# B&R Automation Studio project turbo-parakeet-aka-lab_3
Automation Studio 

## Logical view

### Global.var
```iecst
VAR
	AxisX : ACP10AXIS_typ := (0);
	AxisX_EncIf : SdcEncIf16_typ := (0);
	AxisX_DrvIf : SdcDrvIf16_typ := (0);
	AxisX_DiDoIf : SdcDiDoIf_typ := (0);
	AxisX_HW : SdcHwCfg_typ := (0);
	AxisY : ACP10AXIS_typ := (0);
	AxisY_EncIf : SdcEncIf16_typ := (0);
	AxisY_DrvIf : SdcDrvIf16_typ := (0);
	AxisY_DiDoIf : SdcDiDoIf_typ := (0);
	AxisY_HW : SdcHwCfg_typ := (0);
	AxisZ : ACP10AXIS_typ := (0);
	AxisZ_EncIf : SdcEncIf16_typ := (0);
	AxisZ_DrvIf : SdcDrvIf16_typ := (0);
	AxisZ_DiDoIf : SdcDiDoIf_typ := (0);
	AxisZ_HW : SdcHwCfg_typ := (0);
	gAxis01 : ACP10AXIS_typ := (0);
	gAxis02 : ACP10AXIS_typ := (0);
	gAxisTest : ACP10AXIS_typ := (0);
	gAxisTest_HW : SdcHwCfg_typ := (0);
	gAxisTest_DrvIf : SdcDrvIf16_typ := (0);
	gAxisTest_DiDoIf : SdcDiDoIf_typ := (0);
	gAxisTest_ModuleOk : BOOL := 0;
	gAxis03 : ACP10AXIS_typ := (0);
	gAxis03_HW : SdcHwCfg_typ := (0);
	gAxis03_DrvIf : SdcDrvIf16_typ := (0);
	gAxis03_DiDoIf : SdcDiDoIf_typ := (0);
	gAxis03_ModuleOk : BOOL := 0;
	CNCsys : ARNC0CNC_typ;
	position : INT := 0;
	Myspeed : INT := 0;
END_VAR
```

### Program Logical/SDCAxisCtr

#### Main.c
```c
#include <bur/plctypes.h>

#ifdef _DEFAULT_INCLUDES
	#include <AsDefault.h>
#endif

void increase_counters(void);

void _INIT ProgramInit(void)
{
	//Устанваливаем типы SDC модулей
	AxisX_HW.EncIf1_Typ = ncSDC_ENC16;
	AxisX_HW.DiDoIf_Typ = ncSDC_DIDO;
	AxisX_HW.DrvIf_Typ = ncSDC_DRVSERVO16;

	//Устанавливаем имена переменных
	strcpy(AxisX_HW.EncIf1_Name, "AxisX_EncIf");
	strcpy(AxisX_HW.DrvIf_Name, "AxisX_DrvIf");
	strcpy(AxisX_HW.DiDoIf_Name, "AxisX_DiDoIf");

	//Устанавливаем входы готовности и нормальной работы
	AxisX_EncIf.iEncOK = 1;
	AxisX_DrvIf.iDrvOK = 1;
	AxisX_DrvIf.iStatusEnable = 1;
	AxisX_DiDoIf.iDriveReady = 1;

	fb_controller.dt = 0.002;
	fb_controller.k_i = 0.16;
	fb_controller.k_p = 0.0064;
	fb_controller.max_abs_value = 24.0;

	pwm_period = 200;
}

void _CYCLIC ProgramCyclic(void)
{
	position = AxisX.monitor.s;
	Myspeed = AxisX.monitor.v;
	FB_Axis(&axis_X);
	coil_pwm_value = coil_powered ? 32767 : 0;

	increase_counters();

	//Формирование показаний датчика

	AxisX_EncIf.iActTime = (INT)	AsIOTimeCyclicStart();
	AxisX_EncIf.iActPos = axis_X.counter;
	AxisX_DiDoIf.iPosHwEnd = axis_X.endswitch_a_reached;
	AxisX_DiDoIf.iNegHwEnd = axis_X.endswitch_b_reached;
	fb_controller.in = AxisX_DrvIf.oSetPos;

	if((fb_controller.in<min_task)&&(fb_controller.in>(-min_task))) fb_controller.in = 0;
	fb_controller.in = fb_controller.in * 6500/32767 - axis_X.speed;

	FB_Controller(&fb_controller);

	axis_X.pwm_value = fb_controller.out / 24.0 * 32767;
}

void increase_counters(void)
{
	AxisX_EncIf.iLifeCnt++;
	AxisX_DiDoIf.iLifeCntDriveEnable++;
	AxisX_DiDoIf.iLifeCntDriveReady++;
	AxisX_DiDoIf.iLifeCntNegHwEnd++;
	AxisX_DiDoIf.iLifeCntPosHwEnd++;
	AxisX_DiDoIf.iLifeCntReference++;
	AxisX_DrvIf.iLifeCnt++;
}

void _EXIT ProgramExit(void)
{
	// Insert code here

}
```

### Program Logical/SDCAxisCtr1

#### Main.c
```c
#include <bur/plctypes.h>

#ifdef _DEFAULT_INCLUDES
	#include <AsDefault.h>
#endif

void _INIT ProgramInit(void)
{
	//Устанваливаем типы SDC модулей
	//Устанваливаем типы SDC модулей
	AxisY_HW.EncIf1_Typ = ncSDC_ENC16;
	AxisY_HW.DiDoIf_Typ = ncSDC_DIDO;
	AxisY_HW.DrvIf_Typ = ncSDC_DRVSERVO16;

	//Устанавливаем имена переменных
	strcpy(AxisY_HW.EncIf1_Name, "AxisY_EncIf");
	strcpy(AxisY_HW.DrvIf_Name, "AxisY_DrvIf");
	strcpy(AxisY_HW.DiDoIf_Name, "AxisY_DiDoIf");

	//Устанавливаем входы готовности и нормальной работы
	AxisY_EncIf.iEncOK = 1;
	AxisY_DrvIf.iDrvOK = 1;
	AxisY_DrvIf.iStatusEnable = 1;
	AxisY_DiDoIf.iDriveReady = 1;

	fb_controller.dt = 0.002;
	fb_controller.k_i = 0.16;
	fb_controller.k_p = 0.0064;
	fb_controller.max_abs_value = 24.0;

	pwm_period = 200;

	//Устанавливаем имена переменных

	//Устанавливаем входы готовности и нормальной работы

}

void _CYCLIC ProgramCyclic(void)
{

	FB_Axis(&axis_Y);
	coil_pwm_value = coil_powered ? 32767 : 0;

	increase_counters();

	//Формирование показаний датчика

	AxisY_EncIf.iActTime = (INT)	AsIOTimeCyclicStart();
	AxisY_EncIf.iActPos = axis_Y.counter;
	AxisY_DiDoIf.iPosHwEnd = axis_Y.endswitch_a_reached;
	AxisY_DiDoIf.iNegHwEnd = axis_Y.endswitch_b_reached;
	fb_controller.in = AxisY_DrvIf.oSetPos;

	if((fb_controller.in<min_task)&&(fb_controller.in>(-min_task))) fb_controller.in = 0;
	fb_controller.in = fb_controller.in * 6500/32767 - axis_Y.speed;

	FB_Controller(&fb_controller);

	axis_Y.pwm_value = fb_controller.out / 24.0 * 32767;
	//Формирование показаний датчика

}

void increase_counters(void)
{

		AxisY_EncIf.iLifeCnt++;
		AxisY_DiDoIf.iLifeCntDriveEnable++;
		AxisY_DiDoIf.iLifeCntDriveReady++;
		AxisY_DiDoIf.iLifeCntNegHwEnd++;
		AxisY_DiDoIf.iLifeCntPosHwEnd++;
		AxisY_DiDoIf.iLifeCntReference++;
		AxisY_DrvIf.iLifeCnt++;

}

void _EXIT ProgramExit(void)
{
	// Insert code here

}
```

### Program Logical/SDCAxisCtr2

#### Main.c
```c
#include <bur/plctypes.h>

#ifdef _DEFAULT_INCLUDES
	#include <AsDefault.h>
#endif

void _INIT ProgramInit(void)
{
	//Устанваливаем типы SDC модулей

	//Устанваливаем типы SDC модулей
	AxisZ_HW.EncIf1_Typ = ncSDC_ENC16;
	AxisZ_HW.DiDoIf_Typ = ncSDC_DIDO;
	AxisZ_HW.DrvIf_Typ = ncSDC_DRVSERVO16;

	//Устанавливаем имена переменных
	strcpy(AxisZ_HW.EncIf1_Name, "AxisZ_EncIf");
	strcpy(AxisZ_HW.DrvIf_Name, "AxisZ_DrvIf");
	strcpy(AxisZ_HW.DiDoIf_Name, "AxisZ_DiDoIf");

	//Устанавливаем входы готовности и нормальной работы
	AxisZ_EncIf.iEncOK = 1;
	AxisZ_DrvIf.iDrvOK = 1;
	AxisZ_DrvIf.iStatusEnable = 1;
	AxisZ_DiDoIf.iDriveReady = 1;

	fb_controller.dt = 0.002;
	fb_controller.k_i = 0.16;
	fb_controller.k_p = 0.0064;
	fb_controller.max_abs_value = 24.0;

	pwm_period = 200;
	//Устанавливаем имена переменных

	//Устанавливаем входы готовности и нормальной работы

}

void _CYCLIC ProgramCyclic(void)
{
	FB_Axis(&axis_Z);
	coil_pwm_value = coil_powered ? 32767 : 0;

	increase_counters();

	//Формирование показаний датчика

	AxisZ_EncIf.iActTime = (INT)	AsIOTimeCyclicStart();
	AxisZ_EncIf.iActPos = axis_Z.counter;
	AxisZ_DiDoIf.iPosHwEnd = axis_Z.endswitch_a_reached;
	AxisZ_DiDoIf.iNegHwEnd = axis_Z.endswitch_b_reached;
	fb_controller.in = AxisZ_DrvIf.oSetPos;

	if((fb_controller.in<min_task)&&(fb_controller.in>(-min_task))) fb_controller.in = 0;
	fb_controller.in = fb_controller.in * 6500/32767 - axis_Z.speed;

	FB_Controller(&fb_controller);

	axis_Z.pwm_value = fb_controller.out / 24.0 * 32767;

}

void increase_counters(void)
{
	AxisZ_EncIf.iLifeCnt++;
	AxisZ_DiDoIf.iLifeCntDriveEnable++;
	AxisZ_DiDoIf.iLifeCntDriveReady++;
	AxisZ_DiDoIf.iLifeCntNegHwEnd++;
	AxisZ_DiDoIf.iLifeCntPosHwEnd++;
	AxisZ_DiDoIf.iLifeCntReference++;
	AxisZ_DrvIf.iLifeCnt++;
}

void _EXIT ProgramExit(void)
{
	// Insert code here

}
```
